PROGRAM Safety
VAR
	rTrig : R_Trig;
	tonDelay : TON;
END_VAR


IF TS.iSafetyMat1 AND TS.iSafetyMat2 AND TS.iEStop1 AND TS.iEStop2 THEN
	TS.iSafetyMatAlarm := FALSE;
ELSE
	TS.iSafetyMatAlarm := TRUE;
END_IF



IF NOT TS.iEStop1 OR NOT TS.iEStop2 OR MC.iState = 100 THEN
	TS.oReset := FALSE;
	TS.oErrAckInput := FALSE;
	TS.oErrAckOutput := FALSE;
	TS.oRunInput := FALSE;
	TS.oRunOutput := FALSE;
	//Module_IO.iRelaySwitch := FALSE;
ELSIF Module_IO.iResetButton THEN // Reset button, toggle only
	TS.oErrAckInput := TRUE;
	TS.oErrAckOutput := TRUE;
	//Module_IO.iRelaySwitch := TRUE;
	TS.oRunInput := TRUE;
	TS.oRunOutput := TRUE;
END_IF



(********* Bypass to be used for screens  **********
IF HMI_IO.iDigital[1] THEN //Bypass/Run switch
	TS.oRunInput := TRUE;
	TS.oRunOutput := TRUE;
	HMI_IO.iMotorControl[5] := TRUE;
ELSE
	TS.oRunInput := FALSE;
	TS.oRunOutput := FALSE;
	HMI_IO.iMotorControl[5] := FALSE;
END_IF
    **********************************************)

END_PROGRAM

(* stored: Version 1.1.0.1, ProductVersion 3.1.4024.11
   POU Safety: Id {77b90171-3616-47b4-82e7-fc27d29ea278}, SpecialFunc None *)
